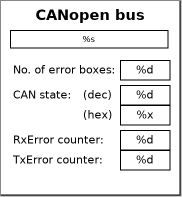
VISUALIZATION VISU_CANopenBus  // 182x197
VAR_IN_OUT
	ref : CANopenBus;
	widget : CANopenBusWidget;
END_VAR
    Rectangle (0,0 180x195)
    Rectangle (0,0 180x30), "CANopen bus"
    Label (10,55 135x30), "No. of error boxes:"
    Rectangle (120,60 50x20), "%d", text variable: ref.error
    Frame (10,30 160x20)
        shows VISU_StatusWidget(widget := widget.actualStatus)
    Label (10,80 155x30), "CAN state:"
    Rectangle (120,85 50x20), "%d", text variable: ref.canState
    Label (80,85 35x20), "(dec)"
    Rectangle (120,105 50x20), "%x", text variable: ref.canState
    Label (80,105 40x20), "(hex)"
    Label (10,125 135x30), "RxError counter:"
    Rectangle (120,130 50x20), "%d", text variable: ref.rxErrorCounter
    Label (10,145 135x30), "TxError counter:"
    Rectangle (120,150 50x20), "%d", text variable: ref.txErrorCounter
END_VISUALIZATION

// ---- MTCS/Common/Visu/VISU_ConfigSINTEntry.TcVIS
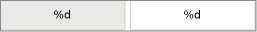
VISUALIZATION VISU_ConfigSINTEntry  // 257x32
VAR_IN_OUT
    active : SINT;
    editable : SINT;
END_VAR
    Textfield (0,0 125x30), "%d", text variable: active, input disabled if: TRUE
    Textfield (130,0 125x30), "%d", text variable: editable, colour toggle: editable <> active
        OnMouseClick: write the text variable via Default
END_VISUALIZATION

// ---- MTCS/Common/Visu/VISU_EtherCatFillerDevice.TcVIS
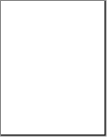
VISUALIZATION VISU_EtherCatFillerDevice  // 107x137
    Rectangle (0,0 105x135)
END_VISUALIZATION

// ---- MTCS/Common/Visu/VISU_AX522DriveChannel.TcVIS
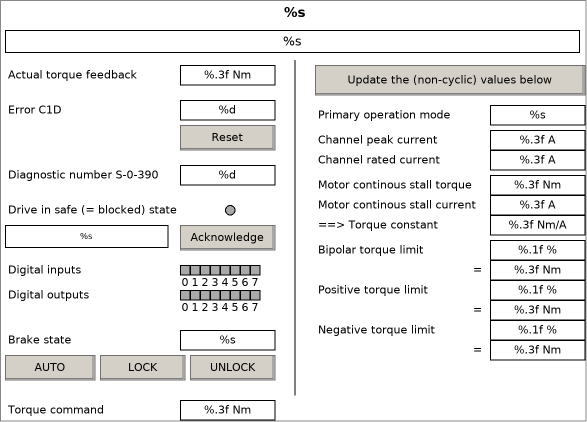
VISUALIZATION VISU_AX522DriveChannel  // 587x422
VAR_IN_OUT
    ref : AX52XXDriveChannel;
    widget : AX52XXDriveChannelWidget;
END_VAR
    Frame (5,30 580x25)
        shows VISU_StatusWidget(widget := widget.actualStatus)
    Rectangle (5,0 580x25), "%s", text variable: widget.name
    Label (315,130 175x20), "Channel peak current"
    Rectangle (490,130 95x20), "%.3f A", text variable: ref.channelPeakCurrent.amps.value
    Label (315,150 175x20), "Channel rated current"
    Rectangle (490,150 95x20), "%.3f A", text variable: ref.channelRatedCurrent.amps.value
    Label (315,175 175x20), "Motor continous stall torque"
    Label (315,195 175x20), "Motor continous stall current"
    Rectangle (490,175 95x20), "%.3f Nm", text variable: ref.continuousStallTorque.newtonmeter.value
    Rectangle (490,195 95x20), "%.3f A", text variable: ref.continuousStallCurrent.amps.value
    Label (315,215 175x20), "==> Torque constant"
    Rectangle (490,215 95x20), "%.3f Nm/A", text variable: ref.torqueConstant
    Button (315,65 270x30), "Update the (non-cyclic) values below", input disabled if: ref.processes.update.statuses.enabledStatus.disabled
        OnMouseClick: execute { ref.processes.update.do_request := TRUE; }
    Label (315,240 175x20), "Bipolar torque limit"
    Rectangle (490,240 95x20), "%.1f %", text variable: ref.bipolarTorqueLimit.percent.value
    Rectangle (490,260 95x20), "%.3f Nm", text variable: ref.bipolarTorqueLimit.newtonmeter.value
    Label (470,260 20x20), "="
    Label (315,280 175x20), "Positive torque limit"
    Rectangle (490,280 95x20), "%.1f %", text variable: ref.positiveTorqueLimit.percent.value
    Rectangle (490,300 95x20), "%.3f Nm", text variable: ref.positiveTorqueLimit.newtonmeter.value
    Label (470,300 20x20), "="
    Label (315,320 175x20), "Negative torque limit"
    Rectangle (490,320 95x20), "%.1f %", text variable: ref.negativeTorqueLimit.percent.value
    Rectangle (490,340 95x20), "%.3f Nm", text variable: ref.negativeTorqueLimit.newtonmeter.value
    Label (470,340 20x20), "="
    Label (5,65 175x20), "Actual torque feedback"
    Rectangle (180,65 95x20), "%.3f Nm", text variable: ref.actualTorqueFeedback.newtonmeter.value
    Label (5,100 175x20), "Error C1D"
    Rectangle (180,100 95x20), "%d", text variable: ref.errorC1D
    Label (5,260 175x20), "Digital inputs"
    Rectangle (180,265 10x10), colour toggle: widget.input0
    Label (180,275 10x15), "0"
    Label (190,275 10x15), "1"
    Label (200,275 10x15), "2"
    Label (210,275 10x15), "3"
    Label (220,275 10x15), "4"
    Label (230,275 10x15), "5"
    Label (240,275 10x15), "6"
    Label (250,275 10x15), "7"
    Rectangle (190,265 10x10), colour toggle: widget.input1
    Rectangle (200,265 10x10), colour toggle: widget.input2
    Rectangle (210,265 10x10), colour toggle: widget.input3
    Rectangle (220,265 10x10), colour toggle: widget.input4
    Rectangle (230,265 10x10), colour toggle: widget.input5
    Rectangle (240,265 10x10), colour toggle: widget.input6
    Rectangle (250,265 10x10), colour toggle: widget.input7
    Label (5,285 175x20), "Digital outputs"
    Rectangle (180,290 10x10), colour toggle: widget.output0
    Label (180,300 10x15), "0"
    Label (190,300 10x15), "1"
    Label (200,300 10x15), "2"
    Label (210,300 10x15), "3"
    Label (220,300 10x15), "4"
    Label (230,300 10x15), "5"
    Label (240,300 10x15), "6"
    Label (250,300 10x15), "7"
    Rectangle (190,290 10x10), colour toggle: widget.output1
    Rectangle (200,290 10x10), colour toggle: widget.output2
    Rectangle (210,290 10x10), colour toggle: widget.output3
    Rectangle (220,290 10x10), colour toggle: widget.output4
    Rectangle (230,290 10x10), colour toggle: widget.output5
    Rectangle (240,290 10x10), colour toggle: widget.output6
    Rectangle (250,290 10x10), colour toggle: widget.output7
    Label (315,105 175x20), "Primary operation mode"
    Rectangle (490,105 95x20), "%s", text variable: ref.operatingMode
    Rectangle (180,330 95x20), "%s", text variable: ref.brakeState
    Label (5,330 175x20), "Brake state"
    Button (5,355 90x25), "AUTO", input disabled if: ref.processes.setBrake.statuses.enabledStatus.disabled
        OnMouseClick: execute { ref.processes.setBrake.set.newState := DriveBrakeStates.BRAKE_AUTOMATIC; ref.processes.setBrake.do_request := TRUE; }
    Button (100,355 85x25), "LOCK", input disabled if: ref.processes.setBrake.statuses.enabledStatus.disabled
        OnMouseClick: execute { ref.processes.setBrake.set.newState := DriveBrakeStates.BRAKE_FORCE_LOCK; ref.processes.setBrake.do_request := TRUE; }
    Button (190,355 85x25), "UNLOCK", input disabled if: ref.processes.setBrake.statuses.enabledStatus.disabled
        OnMouseClick: execute { ref.processes.setBrake.set.newState := DriveBrakeStates.BRAKE_FORCE_UNLOCK; ref.processes.setBrake.do_request := TRUE; }
    Line (295,395) (295,60)
    Button (180,125 95x25), "Reset", input disabled if: ref.processes.reset.statuses.enabledStatus.disabled
        OnMouseClick: execute { ref.processes.reset.do_request := TRUE; }
    Label (5,400 175x20), "Torque command", invisible if: ref.operatingMode <> DriveOperatingModes.OPERATING_MODE_TORQUE_CONTROL
    Rectangle (180,400 95x20), "%.3f Nm", text variable: ref.torqueCommand.newtonmeter.value, invisible if: ref.operatingMode <> DriveOperatingModes.OPERATING_MODE_TORQUE_CONTROL
    Label (5,165 175x20), "Diagnostic number S-0-390"
    Rectangle (180,165 95x20), "%d", text variable: ref.diagnosticNumber
    Label (5,200 215x20), "Drive in safe (= blocked) state"
    Frame (225,200 35x25)
        shows VISU_State_gray_red(state := ref.isInSafetate)
    Button (180,225 95x25), "Acknowledge", input disabled if: ref.processes.acknowledgeSafetyError.statuses.enabledStatus.disabled
        OnMouseClick: execute { ref.processes.acknowledgeSafetyError.do_request := TRUE; }
    Frame (5,225 165x25)
        shows VISU_StatusWidget(widget := widget.processes_acknowledgeSafetyError)
END_VISUALIZATION

// ---- MTCS/Common/Visu/VISU_FaulhaberDriveConfig.TcVIS
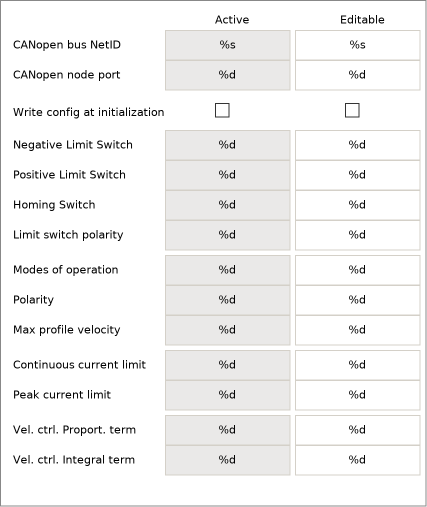
VISUALIZATION VISU_FaulhaberDriveConfig  // 427x507
VAR_IN_OUT
	active : FaulhaberDriveConfig;
	editable : FaulhaberDriveConfig;
END_VAR
    Frame (5,30 415x130)
        shows VISU_FaulhaberDriveConfig_General(active := active, editable := editable)
        shows VISU_FaulhaberDriveConfig_Control(active := active, editable := editable)
        shows VISU_FaulhaberDriveConfig_LimitSwitches(active := active, editable := editable)
    Frame (5,255 415x250)
        shows VISU_FaulhaberDriveConfig_Control(active := active, editable := editable)
        shows VISU_FaulhaberDriveConfig_LimitSwitches(active := active, editable := editable)
        p1986482694: active
        p3357690139: editable
    Frame (5,130 415x140)
        shows VISU_FaulhaberDriveConfig_LimitSwitches(active := active, editable := editable)
        shows VISU_FaulhaberDriveConfig_Control(active := active, editable := editable)
        p1340763843: active
        p1371549466: editable
    Label (170,10 125x20), "Active"
    Label (300,10 125x20), "Editable"
END_VISUALIZATION

// ---- MTCS/Common/Visu/VISU_FaulhaberDrive.TcVIS
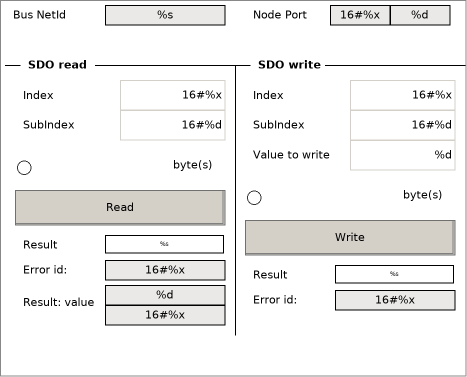
VISUALIZATION VISU_FaulhaberDrive  // 467x377
VAR_IN_OUT
	drive : FaulhaberDrive;
    widget : FaulhaberDriveWidget;
END_VAR
    Frame (0,55 250x320)
        shows VISU_FaulhaberDrive_SDORead(drive := drive, widget := widget)
    Label (10,0 80x30), "Bus NetId"
    Rectangle (105,5 120x20), "%s", text variable: drive.config.CANopenBusNetId
    Rectangle (330,5 60x20), "16#%x", text variable: drive.config.CANopenNodePort
    Label (250,0 80x30), "Node Port"
    Rectangle (390,5 60x20), "%d", text variable: drive.config.CANopenNodePort
    Frame (230,55 235x260)
        shows VISU_FaulhaberDrive_SDOWrite(drive := drive, widget := widget)
    Line (235,65) (235,335)
END_VISUALIZATION

// ---- MTCS/Common/Visu/VISU_ConfigStringEntry.TcVIS
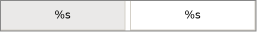
VISUALIZATION VISU_ConfigStringEntry  // 257x32
VAR_IN_OUT
    active : STRING;
    editable : STRING;
END_VAR
    Textfield (0,0 125x30), "%s", text variable: active, input disabled if: TRUE
    Textfield (130,0 125x30), "%s", text variable: editable, colour toggle: editable <> active
        OnMouseClick: write the text variable via Default
END_VISUALIZATION

// ---- MTCS/Common/Visu/VISU_FaulhaberDriveConfig_LimitSwitches.TcVIS
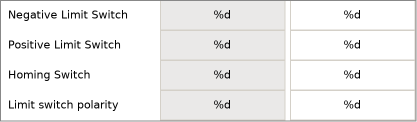
VISUALIZATION VISU_FaulhaberDriveConfig_LimitSwitches  // 417x122
VAR_IN_OUT
	active : FaulhaberDriveConfig;
	editable : FaulhaberDriveConfig;
END_VAR
    Label (5,0 135x30), "Negative Limit Switch"
    Frame (160,0 255x30)
        shows VISU_ConfigUSINTEntry(active := active.negativeLimitSwitch, editable := editable.negativeLimitSwitch)
    Label (5,30 135x30), "Positive Limit Switch"
    Frame (160,30 255x30)
        shows VISU_ConfigUSINTEntry(active := active.positiveLimitSwitch, editable := editable.positiveLimitSwitch)
    Label (5,60 135x30), "Homing Switch"
    Frame (160,60 255x30)
        shows VISU_ConfigUSINTEntry(active := active.homingSwitch, editable := editable.homingSwitch)
    Frame (160,90 255x30)
        shows VISU_ConfigUSINTEntry(active := active.limitSwitchPolarity, editable := editable.limitSwitchPolarity)
    Label (5,90 155x30), "Limit switch polarity"
END_VISUALIZATION

// ---- MTCS/Common/Visu/VISU_FaulhaberDriveConfig_General.TcVIS
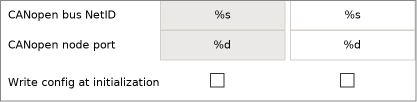
VISUALIZATION VISU_FaulhaberDriveConfig_General  // 417x102
VAR_IN_OUT
	active : FaulhaberDriveConfig;
	editable : FaulhaberDriveConfig;
END_VAR
    Label (5,0 125x30), "CANopen bus NetID"
    Frame (160,0 175x30)
        shows VISU_ConfigStringEntry(active := active.CANopenBusNetId, editable := editable.CANopenBusNetId)
    Label (5,30 125x30), "CANopen node port"
    Frame (160,30 175x30)
        shows VISU_ConfigUINTEntry(active := active.CANopenNodePort, editable := editable.CANopenNodePort)
    Frame (160,65 255x30)
        shows VISU_ConfigBOOLEntry(active := active.sendAtInitialization, editable := editable.sendAtInitialization)
    Label (5,65 155x35), "Write config at initialization"
END_VISUALIZATION

// ---- MTCS/Common/Visu/VISU_FaulhaberDriveConfig_Control.TcVIS
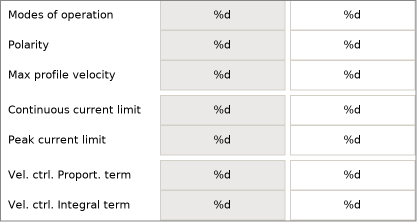
VISUALIZATION VISU_FaulhaberDriveConfig_Control  // 417x222
VAR_IN_OUT
	active : FaulhaberDriveConfig;
	editable : FaulhaberDriveConfig;
END_VAR
    Label (5,30 135x30), "Polarity"
    Frame (160,95 175x30)
        shows VISU_ConfigUINTEntry(active := active.continuousCurrentLimit, editable := editable.continuousCurrentLimit)
    Label (5,95 135x30), "Continuous current limit"
    Label (5,125 135x30), "Peak current limit"
    Frame (160,125 175x30)
        shows VISU_ConfigUINTEntry(active := active.peakCurrentLimit, editable := editable.peakCurrentLimit)
    Frame (160,160 175x30)
        shows VISU_ConfigUINTEntry(active := active.velocityControlProportionalTerm, editable := editable.velocityControlProportionalTerm)
    Label (5,160 135x30), "Vel. ctrl. Proport. term"
    Label (5,190 135x30), "Vel. ctrl. Integral term"
    Frame (160,190 175x30)
        shows VISU_ConfigUINTEntry(active := active.velocityControlIntegralTerm, editable := editable.velocityControlIntegralTerm)
    Label (5,0 135x30), "Modes of operation"
    Frame (160,0 255x30)
        shows VISU_ConfigUSINTEntry(active := active.modesOfOperation, editable := editable.modesOfOperation)
    Frame (160,30 255x30)
        shows VISU_ConfigUSINTEntry(active := active.polarity, editable := editable.polarity)
    Frame (160,60 255x30)
        shows VISU_ConfigUDINTEntry(active := active.maxProfileVelocity, editable := editable.maxProfileVelocity)
    Label (5,60 135x30), "Max profile velocity"
END_VISUALIZATION

// ---- MTCS/Common/Visu/VISU_FaulhaberDrive_SDOWrite.TcVIS
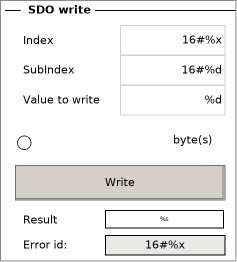
VISUALIZATION VISU_FaulhaberDrive_SDOWrite  // 237x262
VAR_IN_OUT
	drive : FaulhaberDrive;
    widget : FaulhaberDriveWidget;
END_VAR
    Textfield (120,85 105x30), "%d", text variable: drive.processes.write.set.value4Bytes, invisible if: widget.writeNoOfBytes <> 4, input disabled if: drive.processes.write.statuses.enabledStatus.disabled
        OnMouseClick: write the text variable via VisuDialogs.Numpad
    Textfield (120,85 105x30), "%d", text variable: drive.processes.write.set.value2Bytes, invisible if: widget.writeNoOfBytes <> 2, input disabled if: drive.processes.write.statuses.enabledStatus.disabled
        OnMouseClick: write the text variable via VisuDialogs.Numpad
    Textfield (120,85 105x30), "%d", text variable: drive.processes.write.set.value1Byte, invisible if: widget.writeNoOfBytes <> 1, input disabled if: drive.processes.write.statuses.enabledStatus.disabled
        OnMouseClick: write the text variable via Default
    Label (20,26 100x29), "Index"
    Button (15,165 210x35), "Write", input disabled if: drive.processes.write.statuses.enabledStatus.disabled
        OnMouseClick: execute { drive.processes.write.set.noOfBytes := widget.writeNoOfBytes; drive.processes.write.do_request := TRUE; }
    Textfield (120,55 105x30), "16#%d", text variable: drive.processes.write.set.subindex, input disabled if: drive.processes.write.statuses.enabledStatus.disabled
        OnMouseClick: write the text variable via Default
    Label (20,55 95x30), "SubIndex"
    Line (5,10) (20,10)
    Label (25,0 150x20), "SDO write"
    Line (95,10) (235,10)
    Textfield (120,25 105x30), "16#%x", text variable: drive.processes.write.set.index, input disabled if: drive.processes.write.statuses.enabledStatus.disabled
        OnMouseClick: write the text variable via Default
    Frame (105,210 120x20)
        shows VISU_StatusWidget(widget := widget.sdoWriteStatus)
    RadioButton (15,125 155x35), variable: widget.writeNoOfBytesRadioButtonItem, input disabled if: drive.processes.write.statuses.enabledStatus.disabled
        Areas[0]: Text=1
        Areas[1]: Text=2
        Areas[2]: Text=4
    Label (170,125 55x30), "byte(s)"
    Label (20,205 80x30), "Result"
    Rectangle (105,235 120x20), "16#%x", text variable: drive.processes.write.errorId
    Label (20,230 80x30), "Error id:"
    Label (20,85 100x30), "Value to write"
END_VISUALIZATION

// ---- MTCS/Common/Visu/VISU_HiHiLoLoAlarmConfig.TcVIS
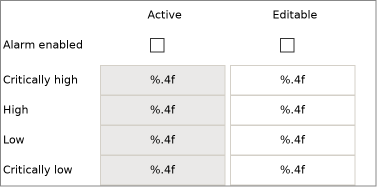
VISUALIZATION VISU_HiHiLoLoAlarmConfig  // 377x187
VAR_IN_OUT
	active : HiHiLoLoAlarmConfig;
    editable : HiHiLoLoAlarmConfig;
END_VAR
    Label (0,30 135x30), "Alarm enabled"
    Frame (100,30 265x30)
        shows VISU_ConfigBOOLEntry(active := active.enabled, editable := editable.enabled)
    Label (0,65 105x30), "Critically high"
    Frame (100,65 275x30)
        shows VISU_ConfigLREAL4Entry(active := active.hiHi, editable := editable.hiHi)
    Label (0,95 105x30), "High"
    Frame (100,95 275x30)
        shows VISU_ConfigLREAL4Entry(active := active.hi, editable := editable.hi)
    Label (0,125 105x30), "Low"
    Frame (100,125 275x30)
        shows VISU_ConfigLREAL4Entry(active := active.lo, editable := editable.lo)
    Label (0,155 105x30), "Critically low"
    Frame (100,155 275x30)
        shows VISU_ConfigLREAL4Entry(active := active.loLo, editable := editable.loLo)
    Label (100,0 130x30), "Active"
    Label (230,0 130x30), "Editable"
END_VISUALIZATION

// ---- MTCS/Common/Visu/VISU_IncrementalEncoder.TcVIS
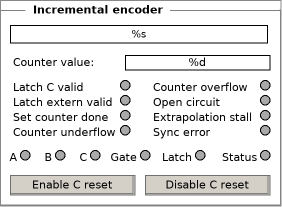
VISUALIZATION VISU_IncrementalEncoder  // 282x207
VAR_IN_OUT
	ref : IncrementalEncoder;
    widget : IncrementalEncoderWidget;
END_VAR
    Polyline (170,10) (280,10) (280,205) (0,205) (0,10) (25,10)
    Label (30,0 150x20), "Incremental encoder"
    Frame (10,25 260x20)
        shows VISU_StatusWidget(widget := widget.actualStatus)
    Label (10,55 105x15), "Counter value:"
    Rectangle (125,55 145x15), "%d", text variable: ref.counterValue
    Label (10,80 105x15), "Latch C valid"
    Frame (120,75 20x20)
        shows VISU_State_gray_green(state := ref.latchCValid)
    Label (10,95 105x15), "Latch extern valid"
    Frame (120,90 20x20)
        shows VISU_State_gray_green(state := ref.latchExternValid)
    Label (10,110 105x15), "Set counter done"
    Frame (120,105 20x20)
        shows VISU_State_gray_green(state := ref.setCounterDone)
    Label (10,125 105x15), "Counter underflow"
    Frame (120,120 10x15)
        shows VISU_State_gray_orange(state := ref.counterUnderflow)
    Label (150,80 105x15), "Counter overflow"
    Frame (260,75 10x15)
        shows VISU_State_gray_orange(state := ref.counterOverflow)
    Label (150,95 105x15), "Open circuit"
    Frame (260,90 10x15)
        shows VISU_State_gray_red(state := ref.openCircuit)
    Label (150,110 105x15), "Extrapolation stall"
    Frame (260,105 10x15)
        shows VISU_State_gray_red(state := ref.extrapolationStall)
    Label (150,125 105x15), "Sync error"
    Frame (260,120 10x15)
        shows VISU_State_gray_red(state := ref.syncError)
    Label (0,150 20x15), "A"
    Frame (20,145 15x20)
        shows VISU_State_gray_green(state := ref.statusOfInputA)
    Label (35,150 20x15), "B"
    Label (70,150 20x15), "C"
    Label (100,150 40x15), "Gate"
    Label (155,150 40x15), "Latch"
    Button (10,175 125x20), "Enable C reset", input disabled if: ref.processes.enableCounterResetC.statuses.enabledStatus.disabled
        OnMouseClick: execute { ref.processes.enableCounterResetC.do_request := TRUE; }
    Button (145,175 125x20), "Disable C reset", input disabled if: ref.processes.disableCounterResetC.statuses.enabledStatus.disabled
        OnMouseClick: execute { ref.processes.disableCounterResetC.do_request := TRUE; }
    Frame (55,145 15x20)
        shows VISU_State_gray_green(state := ref.statusOfInputB)
    Frame (90,145 15x20)
        shows VISU_State_gray_green(state := ref.statusOfInputC)
    Frame (140,145 15x20)
        shows VISU_State_gray_green(state := ref.statusOfInputGate)
    Frame (195,145 15x20)
        shows VISU_State_gray_green(state := ref.statusOfExternLatch)
    Label (210,150 50x15), "Status"
    Frame (260,145 15x20)
        shows VISU_State_gray_green(state := ref.statusOfInputStatus)
END_VISUALIZATION

// ---- MTCS/Common/Visu/VISU_LinearAxis.TcVIS
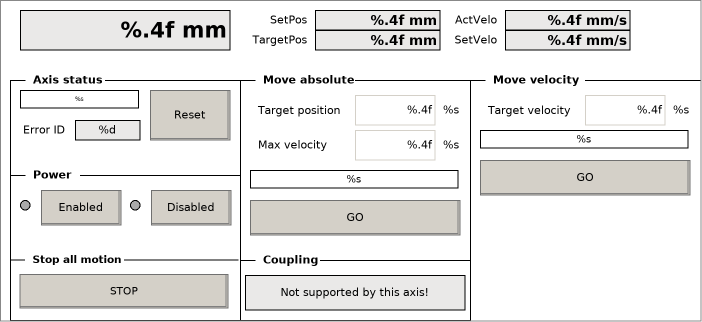
VISUALIZATION VISU_LinearAxis  // 702x322
VAR_IN_OUT
	axis : LinearAxis;
	widget : LinearAxisWidget;
END_VAR
    Rectangle (20,10 210x40), "%.4f mm", text variable: axis.actPos.millimeters.value
    Line (240,80) (240,320)
    Line (10,80) (10,320)
    Line (10,320) (470,320)
    Frame (10,70 230x85)
        shows VISU_BaseAxis_Status(axis := axis, axisWidget := widget.base)
    Frame (10,165 230x60)
        shows VISU_BaseAxis_Power(axis := axis, axisWidget := widget.base)
    Frame (240,70 230x170)
        shows VISU_BaseAxis_MoveAbsolute(axis := axis, axisWidget := widget.base, positionSymbol := widget.positionSymbol, velocitySymbol := widget.velocitySymbol)
    Frame (10,250 230x60)
        shows VISU_BaseAxis_Stop(axis := axis, axisWidget := widget.base)
    Line (470,80) (470,320)
    Frame (240,250 215x60)
        shows VISU_BaseAxis_Gearing(axis := axis, axisWidget := widget.base)
    Frame (470,70 230x125)
        shows VISU_BaseAxis_MoveVelocity(axis := axis, axisWidget := widget.base, positionSymbol := widget.positionSymbol, velocitySymbol := widget.velocitySymbol)
    Rectangle (315,10 125x20), "%.4f mm", text variable: axis.axis_ref.NcToPlc.SetPos
    Label (260,10 50x20), "SetPos"
    Rectangle (315,30 125x20), "%.4f mm", text variable: axis.axis_ref.NcToPlc.TargetPos
    Label (245,30 65x20), "TargetPos"
    Rectangle (505,10 125x20), "%.4f mm/s", text variable: axis.axis_ref.NcToPlc.ActVelo
    Label (450,10 50x20), "ActVelo"
    Label (450,30 50x20), "SetVelo"
    Rectangle (505,30 125x20), "%.4f mm/s", text variable: axis.axis_ref.NcToPlc.SetVelo
END_VISUALIZATION

// ---- MTCS/Common/Visu/VISU_BaseAxis_Stop.TcVIS
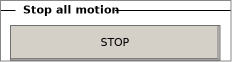
VISUALIZATION VISU_BaseAxis_Stop  // 232x62
VAR_IN_OUT
	axis : BaseAxis;
    axisWidget : BaseAxisWidget;
END_VAR
    Button (10,25 210x35), "STOP", input disabled if: axis.processes.stop.statuses.enabledStatus.disabled
        OnMouseClick: execute { axis.processes.stop.do_request := TRUE; }
    Label (20,0 95x20), "Stop all motion"
    Line (115,10) (230,10)
    Line (0,10) (15,10)
END_VISUALIZATION

// ---- MTCS/Common/Visu/VISU_FaulhaberDrive_SDORead.TcVIS
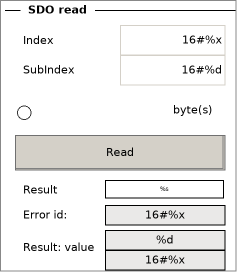
VISUALIZATION VISU_FaulhaberDrive_SDORead  // 237x272
VAR_IN_OUT
	drive : FaulhaberDrive;
    widget : FaulhaberDriveWidget;
END_VAR
    Label (20,26 100x29), "Index"
    Button (15,135 210x35), "Read", input disabled if: drive.processes.read.statuses.enabledStatus.disabled
        OnMouseClick: execute { drive.processes.read.set.noOfBytes := widget.readNoOfBytes; drive.processes.read.do_request := TRUE; }
    Textfield (120,55 105x30), "16#%d", text variable: drive.processes.read.set.subindex, input disabled if: drive.processes.read.statuses.enabledStatus.disabled
        OnMouseClick: write the text variable via Default
    Label (20,55 100x30), "SubIndex"
    Line (5,10) (20,10)
    Label (25,0 150x20), "SDO read"
    Line (95,10) (235,10)
    Textfield (120,25 105x30), "16#%x", text variable: drive.processes.read.set.index, input disabled if: drive.processes.read.statuses.enabledStatus.disabled
        OnMouseClick: write the text variable via Default
    Frame (105,180 120x20)
        shows VISU_StatusWidget(widget := widget.sdoReadStatus)
    RadioButton (15,95 155x35), variable: widget.readNoOfBytesRadioButtonItem, input disabled if: drive.processes.read.statuses.enabledStatus.disabled
        Areas[0]: Text=1
        Areas[1]: Text=2
        Areas[2]: Text=4
    Label (170,95 55x30), "byte(s)"
    Label (20,175 80x30), "Result"
    Label (20,225 80x45), "Result: value"
    Rectangle (105,230 120x20), "%d", text variable: widget.readResultValue
    Rectangle (105,205 120x20), "16#%x", text variable: drive.processes.read.errorId
    Label (20,200 80x30), "Error id:"
    Rectangle (105,250 120x20), "16#%x", text variable: widget.readResultValue
END_VISUALIZATION

// ---- MTCS/Common/Visu/VISU_BaseAxis_MoveAbsolute.TcVIS
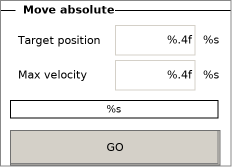
VISUALIZATION VISU_BaseAxis_MoveAbsolute  // 232x167
VAR_IN_OUT
	axis : BaseAxis;
    axisWidget : BaseAxisWidget;
    positionSymbol : STRING;
    velocitySymbol : STRING;
END_VAR
    Label (15,26 100x29), "Target position"
    Button (10,130 210x35), "GO", input disabled if: axis.processes.moveAbsolute.statuses.enabledStatus.disabled
        OnMouseClick: execute { axis.processes.moveAbsolute.do_request := TRUE; }
    Textfield (115,60 80x30), "%.4f", text variable: axis.processes.moveAbsolute.set.maxVelocity, input disabled if: axis.processes.moveAbsolute.statuses.enabledStatus.disabled
        OnMouseClick: write the text variable via VisuDialogs.Numpad
    Label (15,60 100x30), "Max velocity"
    Line (0,10) (15,10)
    Label (20,0 150x20), "Move absolute"
    Line (115,10) (230,10)
    Textfield (115,25 80x30), "%.4f", text variable: axis.processes.moveAbsolute.set.position, input disabled if: axis.processes.moveAbsolute.statuses.enabledStatus.disabled
        OnMouseClick: write the text variable via VisuDialogs.Numpad
    Frame (10,100 210x20)
        shows VISU_StatusWidget(widget := axisWidget.moveAbsoluteProcess.actualStatus)
    Rectangle (200,25 30x30), "%s", text variable: positionSymbol
    Rectangle (200,60 30x30), "%s", text variable: velocitySymbol
END_VISUALIZATION

// ---- MTCS/Common/Visu/VISU_BaseAxis_Power.TcVIS
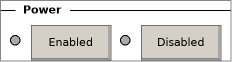
VISUALIZATION VISU_BaseAxis_Power  // 232x62
VAR_IN_OUT
	axis : BaseAxis;
    axisWidget : BaseAxisWidget;
END_VAR
    Button (141,25 80x35), "Disabled", input disabled if: axis.processes.power.statuses.enabledStatus.disabled
        OnMouseClick: execute { axis.processes.power.set.enable := FALSE; axis.processes.power.do_request := TRUE; }
    Frame (120,30 20x20)
        shows VISU_State_gray_orange(state := axis.statuses.poweredStatus.disabled)
    Button (31,25 80x35), "Enabled", input disabled if: axis.processes.power.statuses.enabledStatus.disabled
        OnMouseClick: execute { axis.processes.power.set.enable := TRUE; axis.processes.power.do_request := TRUE; }
    Frame (10,30 25x30)
        shows VISU_State_gray_green(state := axis.statuses.poweredStatus.enabled)
    Label (20,0 55x20), "Power"
    Line (70,10) (230,10)
    Line (0,10) (15,10)
END_VISUALIZATION

// ---- MTCS/Common/Visu/VISU_BaseAxis_Status.TcVIS
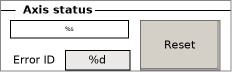
VISUALIZATION VISU_BaseAxis_Status  // 232x72
VAR_IN_OUT
	axis : BaseAxis;
    axisWidget : BaseAxisWidget;
END_VAR
    Label (20,0 75x20), "Axis status"
    Line (95,10) (230,10)
    Line (0,10) (15,10)
    Frame (10,20 120x20)
        shows VISU_StatusWidget(widget := axisWidget.actualStatus)
    Label (10,50 65x20), "Error ID"
    Rectangle (65,50 65x20), "%d", text variable: axis.axis_ref.Status.ErrorId
    Button (140,20 80x50), "Reset", input disabled if: axis.processes.reset.statuses.enabledStatus.disabled
        OnMouseClick: execute { axis.processes.reset.do_request := TRUE; }
END_VISUALIZATION

// ---- MTCS/Common/Visu/VISU_ConfigManager.TcVIS
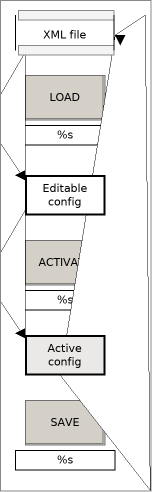
VISUALIZATION VISU_ConfigManager  // 152x492
VAR_IN_OUT
	mgr : ConfigManager;
    widget : ConfigManagerWidget;
END_VAR
    Button (25,75 80x45), "LOAD", input disabled if: mgr.processes.load.statuses.enabledStatus.disabled
        OnMouseClick: execute { mgr.processes.load.do_request := TRUE; }
    Button (25,240 80x45), "ACTIVATE", input disabled if: mgr.processes.activate.statuses.enabledStatus.disabled
        OnMouseClick: execute { mgr.processes.activate.do_request := TRUE; }
    Rectangle (15,125 100x20), "%s", text variable: widget.load.description, colour variable: widget.load.bgColor
        p55702900: widget.load.fgColor
    Rectangle (15,290 100x20), "%s", text variable: widget.load.description, colour variable: widget.load.bgColor
        p55702900: widget.load.fgColor
    Button (25,400 80x45), "SAVE", input disabled if: mgr.processes.save.statuses.enabledStatus.disabled
        OnMouseClick: execute { mgr.processes.save.do_request := TRUE; }
    Rectangle (15,450 100x20), "%s", text variable: widget.save.description, colour variable: widget.save.bgColor
        p55702900: widget.load.fgColor
    Polygon (25,52) (0,95) (-5,135) (25,180)
    Polygon (15,175) (25,170) (25,180)
    Polygon (25,210) (0,253) (-5,293) (25,338)
    Polygon (15,333) (25,328) (25,338)
    Polygon (60,375) (150,490) (145,15) (115,35)
    Polygon (115,35) (125,35) (120,45)
    RoundedRectangle (25,175 80x40), "Editable config"
    Pie (18,45 96x10)
    Pie (18,10 96x10)
    Line (114,50) (114,15)
    RoundedRectangle (25,335 80x40), "Active config"
    Label (20,20 90x30), "XML file"
    Line (15,15) (15,50)
END_VISUALIZATION

// ---- MTCS/Common/Visu/VISU_EtherCatDevice.TcVIS
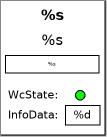
VISUALIZATION VISU_EtherCatDevice  // 107x137
VAR_IN_OUT
	device : EtherCatDevice;
	widget : EtherCatDeviceWidget;
END_VAR
    Rectangle (0,0 105x135)
    Rectangle (0,0 105x30), "%s", text variable: device.typeId
    Rectangle (0,25 105x30), "%s", text variable: device.id
    Label (5,80 60x30), "WcState:"
    Label (5,100 60x30), "InfoData:"
    Rectangle (65,105 35x20), "%d", text variable: device.infoData
    Frame (5,55 95x20)
        shows VISU_StatusWidget(widget := widget.actualStatus)
    Frame (75,85 15x15)
        shows VISU_State_green_red(state := device.wcState)
END_VISUALIZATION

// ---- MTCS/Common/Visu/VISU_Measurement.TcVIS
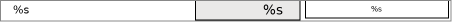
VISUALIZATION VISU_Measurement  // 452x22
VAR_IN_OUT
    widget : MeasurementWidget;
END_VAR
    Rectangle (10,0 180x20), "%s", text variable: widget.name
    Rectangle (195,0 105x20)
    Frame (305,0 145x20)
        shows VISU_StatusWidget(widget := widget.actualStatusWidget)
    Rectangle (195,0 100x20), "%s", text variable: widget.display
END_VISUALIZATION

// ---- MTCS/Common/Visu/VISU_MeasurementConfig.TcVIS
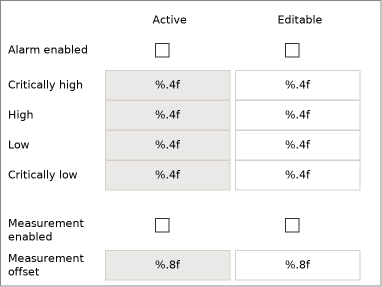
VISUALIZATION VISU_MeasurementConfig  // 382x287
VAR_IN_OUT
	active : MeasurementConfig;
    editable : MeasurementConfig;
END_VAR
    Frame (5,5 375x185)
        shows VISU_HiHiLoLoAlarmConfig(active := active.alarms, editable := editable.alarms)
    Frame (105,210 255x30)
        shows VISU_ConfigBOOLEntry(active := active.enabled, editable := editable.enabled)
    Label (5,210 95x40), "Measurement enabled"
    Label (5,245 95x40), "Measurement offset"
    Frame (105,250 255x30)
        shows VISU_ConfigLREAL8Entry(active := active.offset, editable := editable.offset)
END_VISUALIZATION

// ---- MTCS/Common/Visu/VISU_ProcessStep.TcVIS
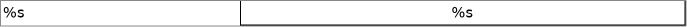
VISUALIZATION VISU_ProcessStep  // 687x27
VAR_IN_OUT
	widget : ProcessStepWidget;
END_VAR
    Rectangle (240,0 445x25), "%s", text variable: widget.statusText, invisible if: widget.inivisible, colour variable: widget.color.bg
        p3450524324: widget.color.fg
        p55702900: widget.color.fg
    Rectangle (0,0 235x25), "%s", text variable: widget.description, invisible if: widget.inivisible
END_VISUALIZATION

// ---- MTCS/Common/Visu/VISU_SimpleRelay.TcVIS
